// LS Electric XG5000 project: 과년1번패턴
// PLC NewPLC
// module base 0 slot 0: 입출력 모듈:XBC-DR20S (DC 24V 입력 12점, 릴레이 출력 8점)

PROGRAM NewProgram (task: 스캔 프로그램)

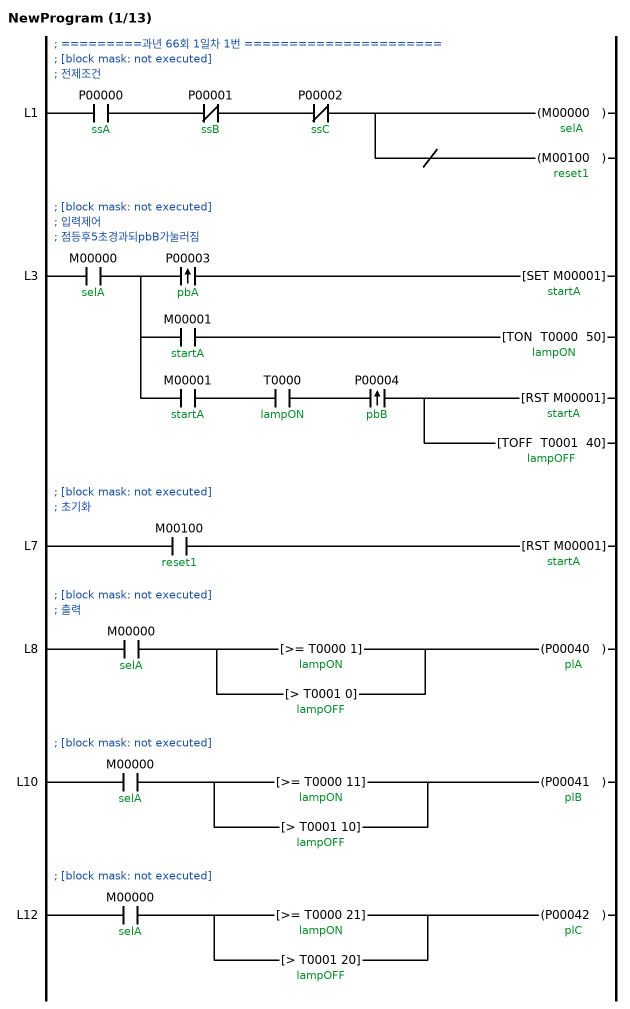
// =========과년 66회 1일차 1번 ======================
; L1 (block mask: not executed)
LOAD      P00000	// ssA
AND NOT   P00001	// ssB
AND NOT   P00002	// ssC
OUT       M00000	// selA
NOT
OUT       M00100	// reset1
// output comment: 전제조건
; L3 (block mask: not executed)
LOAD      M00000	// selA
MPUSH
ANDP      P00003	// pbA
SET       M00001	// startA
MLOAD
AND       M00001	// startA
TON       T0000 50	// lampON
MPOP
AND       M00001	// startA
AND       T0000	// lampON
ANDP      P00004	// pbB
RST       M00001	// startA
TOFF      T0001 40	// lampOFF
// output comment: 입력제어
// output comment: 점등후5초경과되pbB가눌러짐
; L7 (block mask: not executed)
LOAD      M00100	// reset1
RST       M00001	// startA
// output comment: 초기화
; L8 (block mask: not executed)
LOAD      M00000	// selA
LOAD>=    T0000 1	// lampON
OR>       T0001 0	// lampOFF
AND LOAD
OUT       P00040	// plA
// output comment: 출력
; L10 (block mask: not executed)
LOAD      M00000	// selA
LOAD>=    T0000 11	// lampON
OR>       T0001 10	// lampOFF
AND LOAD
OUT       P00041	// plB
; L12 (block mask: not executed)
LOAD      M00000	// selA
LOAD>=    T0000 21	// lampON
OR>       T0001 20	// lampOFF
AND LOAD
OUT       P00042	// plC

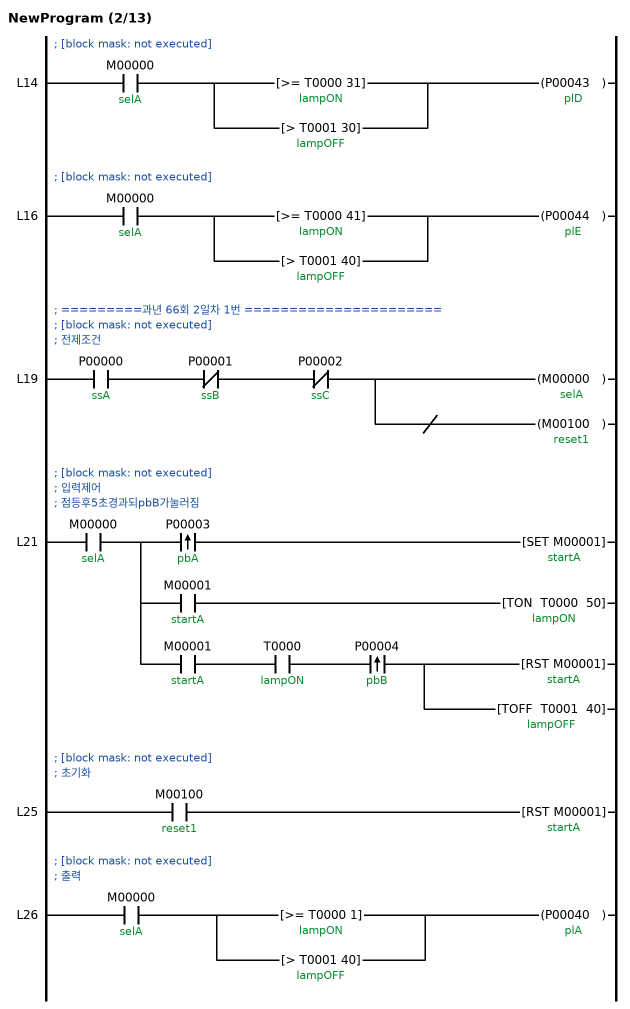
; L14 (block mask: not executed)
LOAD      M00000	// selA
LOAD>=    T0000 31	// lampON
OR>       T0001 30	// lampOFF
AND LOAD
OUT       P00043	// plD
; L16 (block mask: not executed)
LOAD      M00000	// selA
LOAD>=    T0000 41	// lampON
OR>       T0001 40	// lampOFF
AND LOAD
OUT       P00044	// plE
// =========과년 66회 2일차 1번 ======================
; L19 (block mask: not executed)
LOAD      P00000	// ssA
AND NOT   P00001	// ssB
AND NOT   P00002	// ssC
OUT       M00000	// selA
NOT
OUT       M00100	// reset1
// output comment: 전제조건
; L21 (block mask: not executed)
LOAD      M00000	// selA
MPUSH
ANDP      P00003	// pbA
SET       M00001	// startA
MLOAD
AND       M00001	// startA
TON       T0000 50	// lampON
MPOP
AND       M00001	// startA
AND       T0000	// lampON
ANDP      P00004	// pbB
RST       M00001	// startA
TOFF      T0001 40	// lampOFF
// output comment: 입력제어
// output comment: 점등후5초경과되pbB가눌러짐
; L25 (block mask: not executed)
LOAD      M00100	// reset1
RST       M00001	// startA
// output comment: 초기화
; L26 (block mask: not executed)
LOAD      M00000	// selA
LOAD>=    T0000 1	// lampON
OR>       T0001 40	// lampOFF
AND LOAD
OUT       P00040	// plA
// output comment: 출력

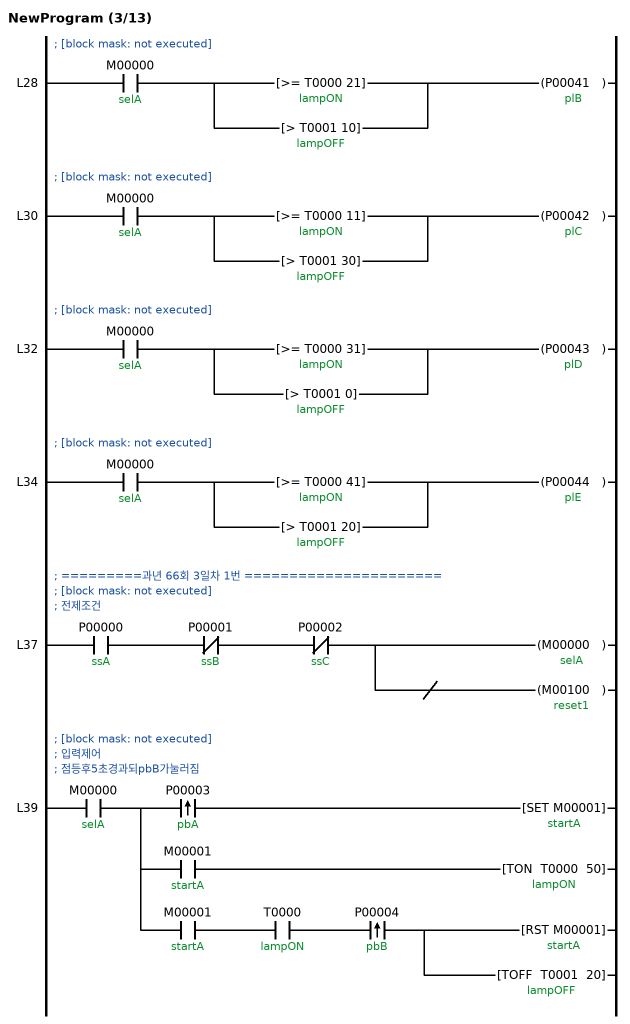
; L28 (block mask: not executed)
LOAD      M00000	// selA
LOAD>=    T0000 21	// lampON
OR>       T0001 10	// lampOFF
AND LOAD
OUT       P00041	// plB
; L30 (block mask: not executed)
LOAD      M00000	// selA
LOAD>=    T0000 11	// lampON
OR>       T0001 30	// lampOFF
AND LOAD
OUT       P00042	// plC
; L32 (block mask: not executed)
LOAD      M00000	// selA
LOAD>=    T0000 31	// lampON
OR>       T0001 0	// lampOFF
AND LOAD
OUT       P00043	// plD
; L34 (block mask: not executed)
LOAD      M00000	// selA
LOAD>=    T0000 41	// lampON
OR>       T0001 20	// lampOFF
AND LOAD
OUT       P00044	// plE
// =========과년 66회 3일차 1번 ======================
; L37 (block mask: not executed)
LOAD      P00000	// ssA
AND NOT   P00001	// ssB
AND NOT   P00002	// ssC
OUT       M00000	// selA
NOT
OUT       M00100	// reset1
// output comment: 전제조건
; L39 (block mask: not executed)
LOAD      M00000	// selA
MPUSH
ANDP      P00003	// pbA
SET       M00001	// startA
MLOAD
AND       M00001	// startA
TON       T0000 50	// lampON
MPOP
AND       M00001	// startA
AND       T0000	// lampON
ANDP      P00004	// pbB
RST       M00001	// startA
TOFF      T0001 20	// lampOFF
// output comment: 입력제어
// output comment: 점등후5초경과되pbB가눌러짐

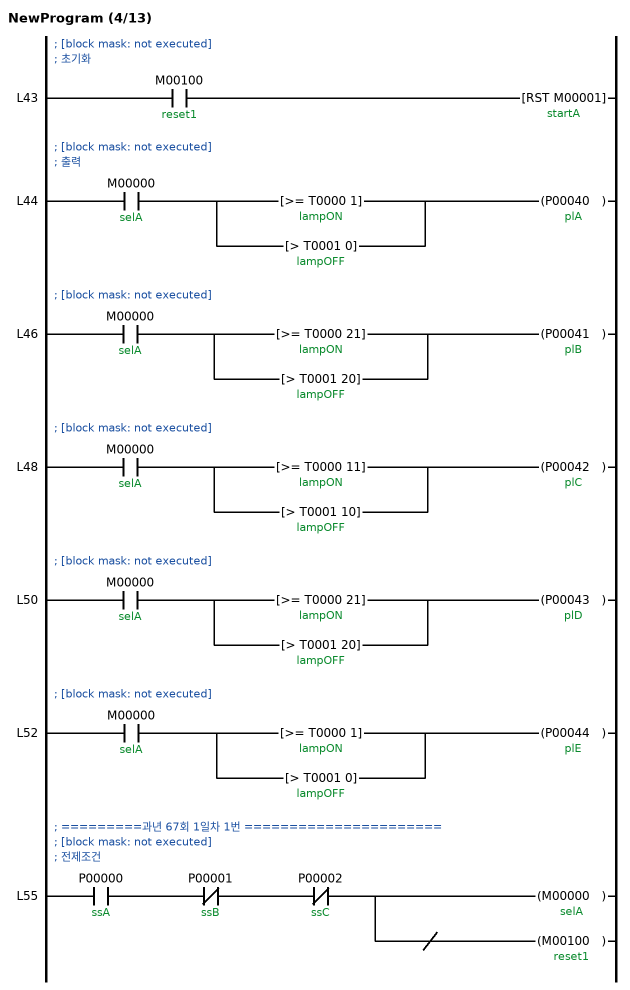
; L43 (block mask: not executed)
LOAD      M00100	// reset1
RST       M00001	// startA
// output comment: 초기화
; L44 (block mask: not executed)
LOAD      M00000	// selA
LOAD>=    T0000 1	// lampON
OR>       T0001 0	// lampOFF
AND LOAD
OUT       P00040	// plA
// output comment: 출력
; L46 (block mask: not executed)
LOAD      M00000	// selA
LOAD>=    T0000 21	// lampON
OR>       T0001 20	// lampOFF
AND LOAD
OUT       P00041	// plB
; L48 (block mask: not executed)
LOAD      M00000	// selA
LOAD>=    T0000 11	// lampON
OR>       T0001 10	// lampOFF
AND LOAD
OUT       P00042	// plC
; L50 (block mask: not executed)
LOAD      M00000	// selA
LOAD>=    T0000 21	// lampON
OR>       T0001 20	// lampOFF
AND LOAD
OUT       P00043	// plD
; L52 (block mask: not executed)
LOAD      M00000	// selA
LOAD>=    T0000 1	// lampON
OR>       T0001 0	// lampOFF
AND LOAD
OUT       P00044	// plE
// =========과년 67회 1일차 1번 ======================
; L55 (block mask: not executed)
LOAD      P00000	// ssA
AND NOT   P00001	// ssB
AND NOT   P00002	// ssC
OUT       M00000	// selA
NOT
OUT       M00100	// reset1
// output comment: 전제조건

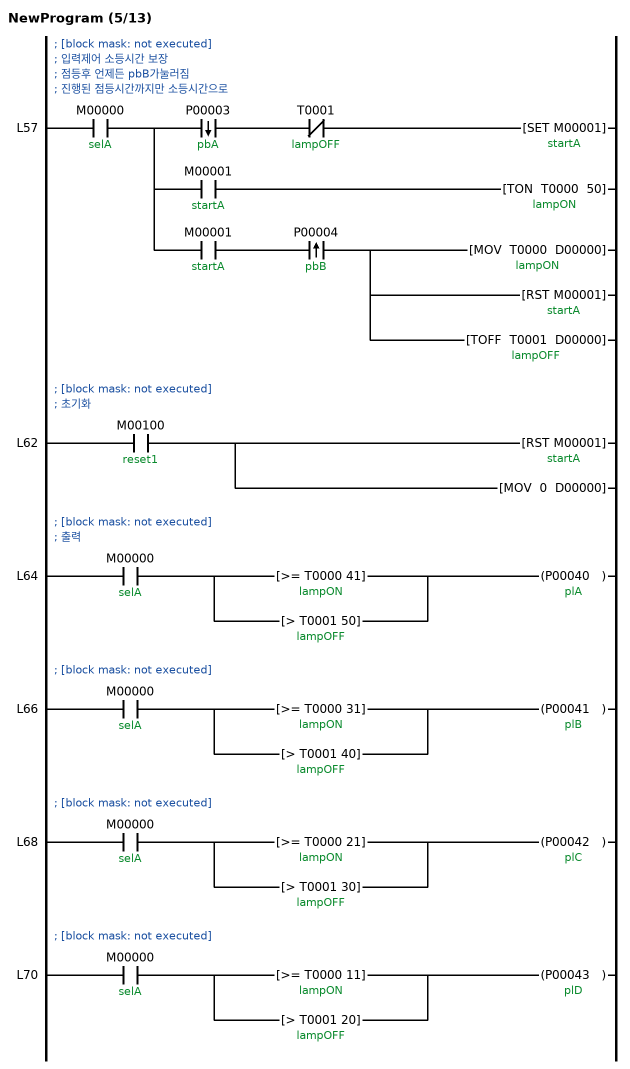
; L57 (block mask: not executed)
LOAD      M00000	// selA
MPUSH
ANDN      P00003	// pbA
AND NOT   T0001	// lampOFF
SET       M00001	// startA
MLOAD
AND       M00001	// startA
TON       T0000 50	// lampON
MPOP
AND       M00001	// startA
ANDP      P00004	// pbB
MOV       T0000 D00000	// lampON
RST       M00001	// startA
TOFF      T0001 D00000	// lampOFF
// output comment: 입력제어 소등시간 보장
// output comment: 점등후 언제든 pbB가눌러짐
// output comment: 
// output comment: 진행된 점등시간까지만 소등시간으로
; L62 (block mask: not executed)
LOAD      M00100	// reset1
RST       M00001	// startA
MOV       0 D00000
// output comment: 초기화
; L64 (block mask: not executed)
LOAD      M00000	// selA
LOAD>=    T0000 41	// lampON
OR>       T0001 50	// lampOFF
AND LOAD
OUT       P00040	// plA
// output comment: 출력
; L66 (block mask: not executed)
LOAD      M00000	// selA
LOAD>=    T0000 31	// lampON
OR>       T0001 40	// lampOFF
AND LOAD
OUT       P00041	// plB
; L68 (block mask: not executed)
LOAD      M00000	// selA
LOAD>=    T0000 21	// lampON
OR>       T0001 30	// lampOFF
AND LOAD
OUT       P00042	// plC
; L70 (block mask: not executed)
LOAD      M00000	// selA
LOAD>=    T0000 11	// lampON
OR>       T0001 20	// lampOFF
AND LOAD
OUT       P00043	// plD

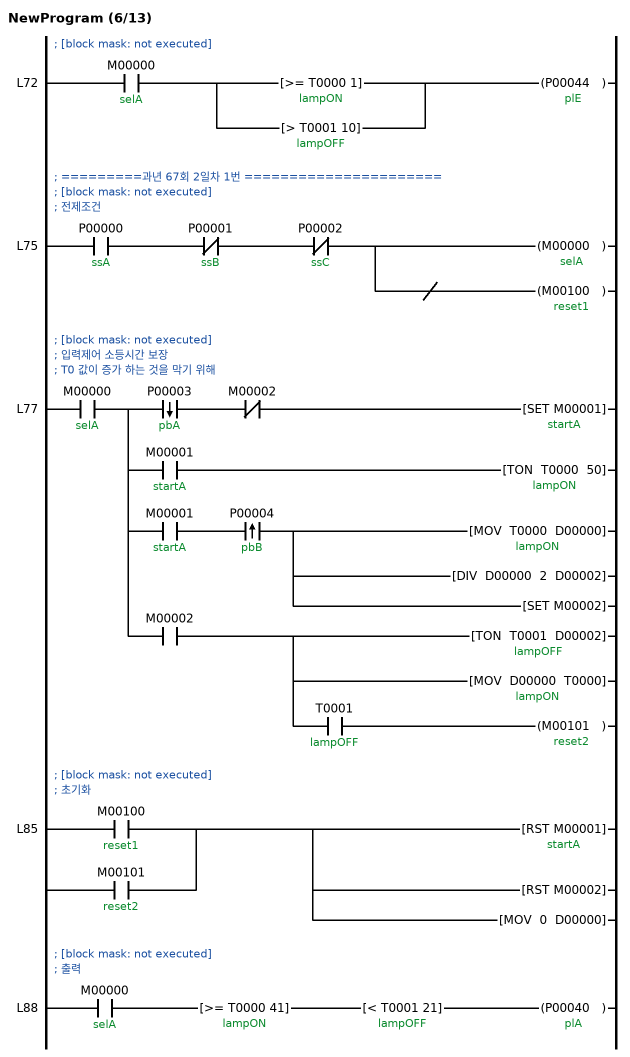
; L72 (block mask: not executed)
LOAD      M00000	// selA
LOAD>=    T0000 1	// lampON
OR>       T0001 10	// lampOFF
AND LOAD
OUT       P00044	// plE
// =========과년 67회 2일차 1번 ======================
; L75 (block mask: not executed)
LOAD      P00000	// ssA
AND NOT   P00001	// ssB
AND NOT   P00002	// ssC
OUT       M00000	// selA
NOT
OUT       M00100	// reset1
// output comment: 전제조건
; L77 (block mask: not executed)
LOAD      M00000	// selA
MPUSH
ANDN      P00003	// pbA
AND NOT   M00002
SET       M00001	// startA
MLOAD
AND       M00001	// startA
TON       T0000 50	// lampON
MLOAD
AND       M00001	// startA
ANDP      P00004	// pbB
MOV       T0000 D00000	// lampON
DIV       D00000 2 D00002
SET       M00002
MPOP
AND       M00002
TON       T0001 D00002	// lampOFF
MOV       D00000 T0000	// lampON
AND       T0001	// lampOFF
OUT       M00101	// reset2
// output comment: 입력제어 소등시간 보장
// output comment: T0 값이 증가 하는 것을 막기 위해
; L85 (block mask: not executed)
LOAD      M00100	// reset1
OR        M00101	// reset2
RST       M00001	// startA
RST       M00002
MOV       0 D00000
// output comment: 초기화
; L88 (block mask: not executed)
LOAD      M00000	// selA
AND>=     T0000 41	// lampON
AND<      T0001 21	// lampOFF
OUT       P00040	// plA
// output comment: 출력

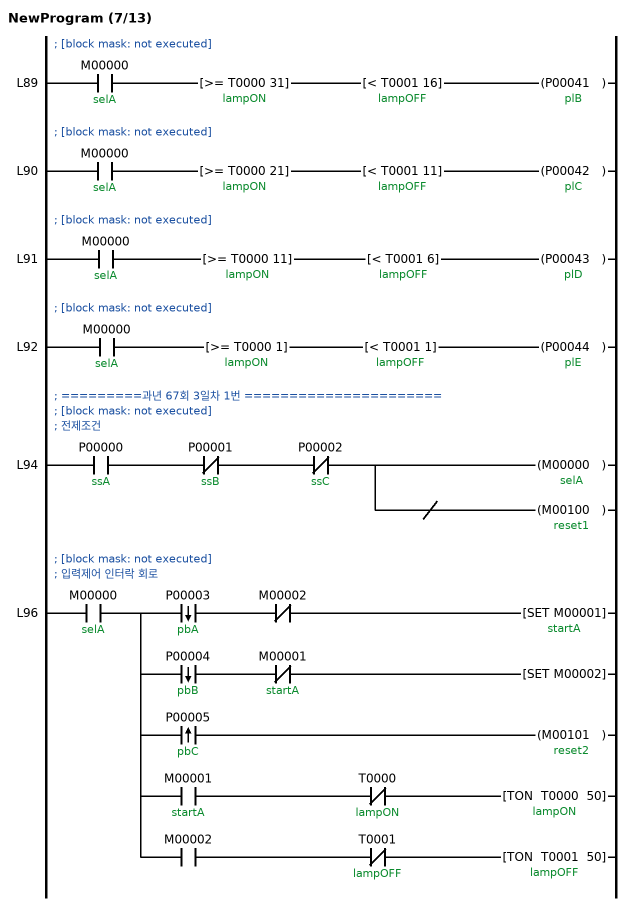
; L89 (block mask: not executed)
LOAD      M00000	// selA
AND>=     T0000 31	// lampON
AND<      T0001 16	// lampOFF
OUT       P00041	// plB
; L90 (block mask: not executed)
LOAD      M00000	// selA
AND>=     T0000 21	// lampON
AND<      T0001 11	// lampOFF
OUT       P00042	// plC
; L91 (block mask: not executed)
LOAD      M00000	// selA
AND>=     T0000 11	// lampON
AND<      T0001 6	// lampOFF
OUT       P00043	// plD
; L92 (block mask: not executed)
LOAD      M00000	// selA
AND>=     T0000 1	// lampON
AND<      T0001 1	// lampOFF
OUT       P00044	// plE
// =========과년 67회 3일차 1번 ======================
; L94 (block mask: not executed)
LOAD      P00000	// ssA
AND NOT   P00001	// ssB
AND NOT   P00002	// ssC
OUT       M00000	// selA
NOT
OUT       M00100	// reset1
// output comment: 전제조건
; L96 (block mask: not executed)
LOAD      M00000	// selA
MPUSH
ANDN      P00003	// pbA
AND NOT   M00002
SET       M00001	// startA
MLOAD
ANDN      P00004	// pbB
AND NOT   M00001	// startA
SET       M00002
MLOAD
ANDP      P00005	// pbC
OUT       M00101	// reset2
MLOAD
AND       M00001	// startA
AND NOT   T0000	// lampON
TON       T0000 50	// lampON
MPOP
AND       M00002
AND NOT   T0001	// lampOFF
TON       T0001 50	// lampOFF
// output comment: 입력제어 인터락 회로

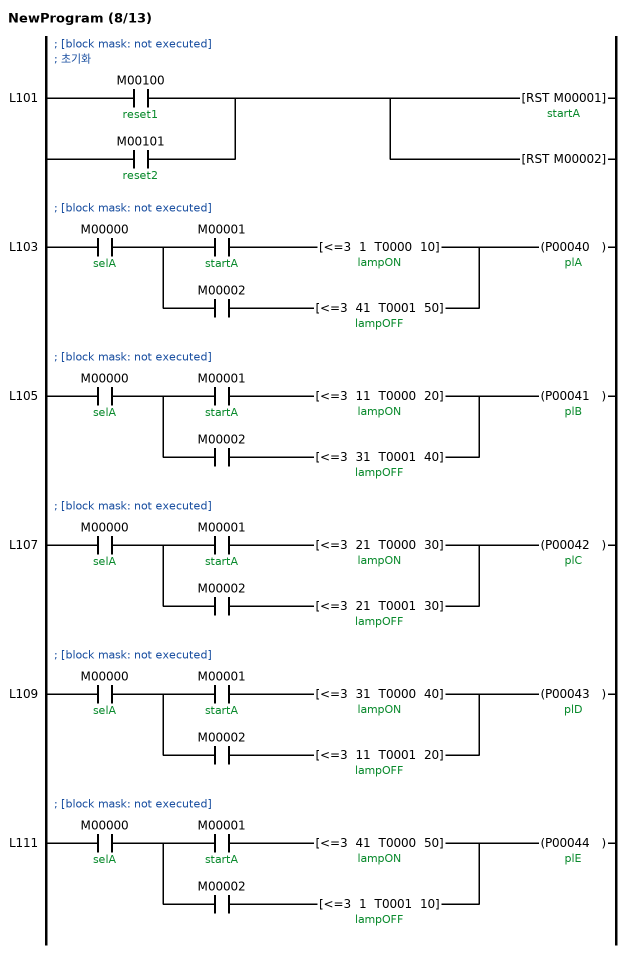
; L101 (block mask: not executed)
LOAD      M00100	// reset1
OR        M00101	// reset2
RST       M00001	// startA
RST       M00002
// output comment: 초기화
; L103 (block mask: not executed)
LOAD      M00000	// selA
LOAD      M00001	// startA
AND<=3    1 T0000 10	// lampON
LOAD      M00002
AND<=3    41 T0001 50	// lampOFF
OR LOAD
AND LOAD
OUT       P00040	// plA
; L105 (block mask: not executed)
LOAD      M00000	// selA
LOAD      M00001	// startA
AND<=3    11 T0000 20	// lampON
LOAD      M00002
AND<=3    31 T0001 40	// lampOFF
OR LOAD
AND LOAD
OUT       P00041	// plB
; L107 (block mask: not executed)
LOAD      M00000	// selA
LOAD      M00001	// startA
AND<=3    21 T0000 30	// lampON
LOAD      M00002
AND<=3    21 T0001 30	// lampOFF
OR LOAD
AND LOAD
OUT       P00042	// plC
; L109 (block mask: not executed)
LOAD      M00000	// selA
LOAD      M00001	// startA
AND<=3    31 T0000 40	// lampON
LOAD      M00002
AND<=3    11 T0001 20	// lampOFF
OR LOAD
AND LOAD
OUT       P00043	// plD
; L111 (block mask: not executed)
LOAD      M00000	// selA
LOAD      M00001	// startA
AND<=3    41 T0000 50	// lampON
LOAD      M00002
AND<=3    1 T0001 10	// lampOFF
OR LOAD
AND LOAD
OUT       P00044	// plE

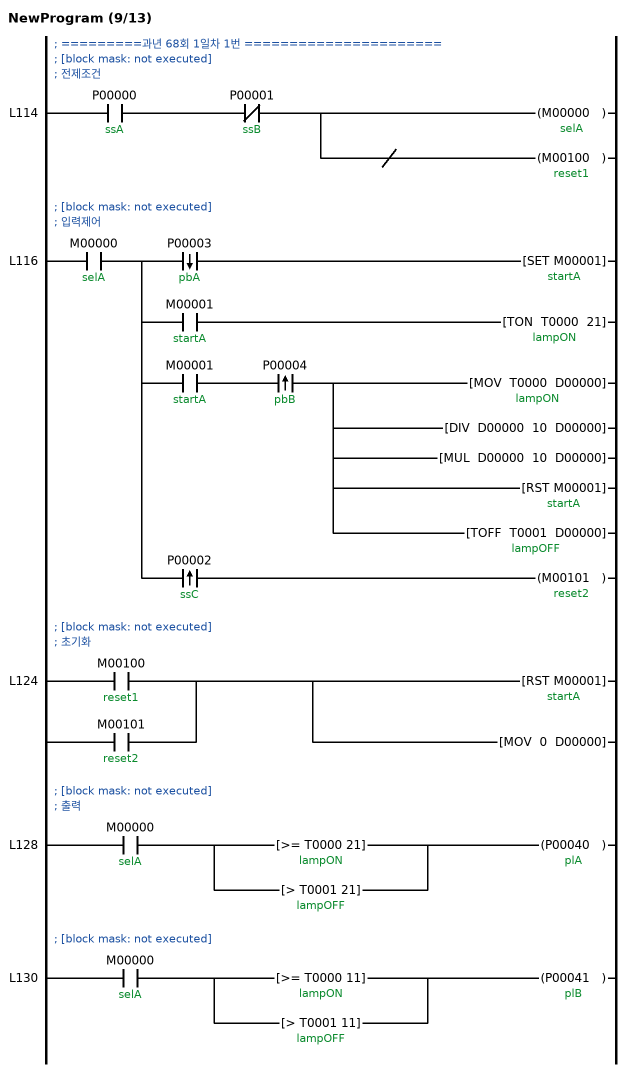
// =========과년 68회 1일차 1번 ======================
; L114 (block mask: not executed)
LOAD      P00000	// ssA
AND NOT   P00001	// ssB
OUT       M00000	// selA
NOT
OUT       M00100	// reset1
// output comment: 전제조건
; L116 (block mask: not executed)
LOAD      M00000	// selA
MPUSH
ANDN      P00003	// pbA
SET       M00001	// startA
MLOAD
AND       M00001	// startA
TON       T0000 21	// lampON
MLOAD
AND       M00001	// startA
ANDP      P00004	// pbB
MOV       T0000 D00000	// lampON
DIV       D00000 10 D00000
MUL       D00000 10 D00000
RST       M00001	// startA
TOFF      T0001 D00000	// lampOFF
MPOP
ANDP      P00002	// ssC
OUT       M00101	// reset2
// output comment: 입력제어
; L124 (block mask: not executed)
LOAD      M00100	// reset1
OR        M00101	// reset2
RST       M00001	// startA
MOV       0 D00000
// output comment: 초기화
; L128 (block mask: not executed)
LOAD      M00000	// selA
LOAD>=    T0000 21	// lampON
OR>       T0001 21	// lampOFF
AND LOAD
OUT       P00040	// plA
// output comment: 출력
; L130 (block mask: not executed)
LOAD      M00000	// selA
LOAD>=    T0000 11	// lampON
OR>       T0001 11	// lampOFF
AND LOAD
OUT       P00041	// plB

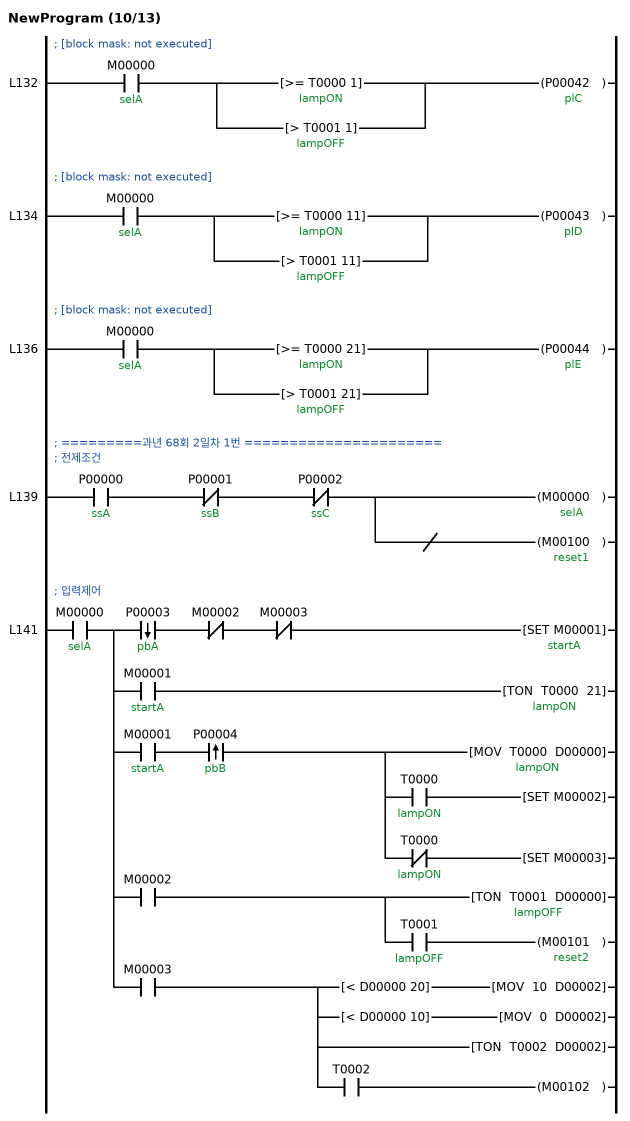
; L132 (block mask: not executed)
LOAD      M00000	// selA
LOAD>=    T0000 1	// lampON
OR>       T0001 1	// lampOFF
AND LOAD
OUT       P00042	// plC
; L134 (block mask: not executed)
LOAD      M00000	// selA
LOAD>=    T0000 11	// lampON
OR>       T0001 11	// lampOFF
AND LOAD
OUT       P00043	// plD
; L136 (block mask: not executed)
LOAD      M00000	// selA
LOAD>=    T0000 21	// lampON
OR>       T0001 21	// lampOFF
AND LOAD
OUT       P00044	// plE
// =========과년 68회 2일차 1번 ======================
; L139
LOAD      P00000	// ssA
AND NOT   P00001	// ssB
AND NOT   P00002	// ssC
OUT       M00000	// selA
NOT
OUT       M00100	// reset1
// output comment: 전제조건
; L141
LOAD      M00000	// selA
MPUSH
ANDN      P00003	// pbA
AND NOT   M00002
AND NOT   M00003
SET       M00001	// startA
MLOAD
AND       M00001	// startA
TON       T0000 21	// lampON
MLOAD
AND       M00001	// startA
ANDP      P00004	// pbB
MOV       T0000 D00000	// lampON
MPUSH
AND       T0000	// lampON
SET       M00002
MPOP
AND NOT   T0000	// lampON
SET       M00003
MLOAD
AND       M00002
TON       T0001 D00000	// lampOFF
AND       T0001	// lampOFF
OUT       M00101	// reset2
MPOP
AND       M00003
MPUSH
AND<      D00000 20
MOV       10 D00002
MLOAD
AND<      D00000 10
MOV       0 D00002
MPOP
TON       T0002 D00002
AND       T0002
OUT       M00102
// output comment: 입력제어

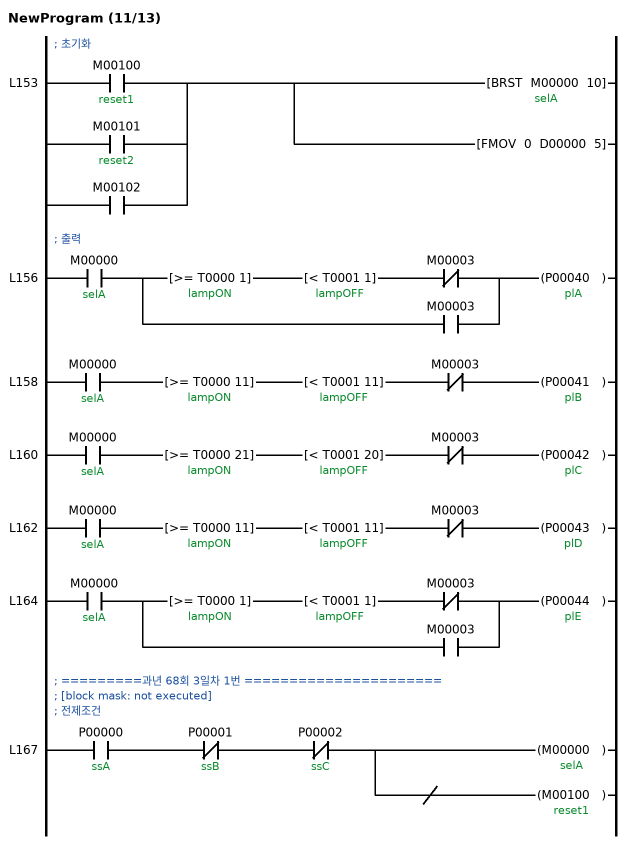
; L153
LOAD      M00100	// reset1
OR        M00101	// reset2
OR        M00102
BRST      M00000 10	// selA
FMOV      0 D00000 5
// output comment: 초기화
; L156
LOAD      M00000	// selA
LOAD>=    T0000 1	// lampON
AND<      T0001 1	// lampOFF
AND NOT   M00003
OR        M00003
AND LOAD
OUT       P00040	// plA
// output comment: 출력
; L158
LOAD      M00000	// selA
AND>=     T0000 11	// lampON
AND<      T0001 11	// lampOFF
AND NOT   M00003
OUT       P00041	// plB
; L160
LOAD      M00000	// selA
AND>=     T0000 21	// lampON
AND<      T0001 20	// lampOFF
AND NOT   M00003
OUT       P00042	// plC
; L162
LOAD      M00000	// selA
AND>=     T0000 11	// lampON
AND<      T0001 11	// lampOFF
AND NOT   M00003
OUT       P00043	// plD
; L164
LOAD      M00000	// selA
LOAD>=    T0000 1	// lampON
AND<      T0001 1	// lampOFF
AND NOT   M00003
OR        M00003
AND LOAD
OUT       P00044	// plE
// =========과년 68회 3일차 1번 ======================
; L167 (block mask: not executed)
LOAD      P00000	// ssA
AND NOT   P00001	// ssB
AND NOT   P00002	// ssC
OUT       M00000	// selA
NOT
OUT       M00100	// reset1
// output comment: 전제조건

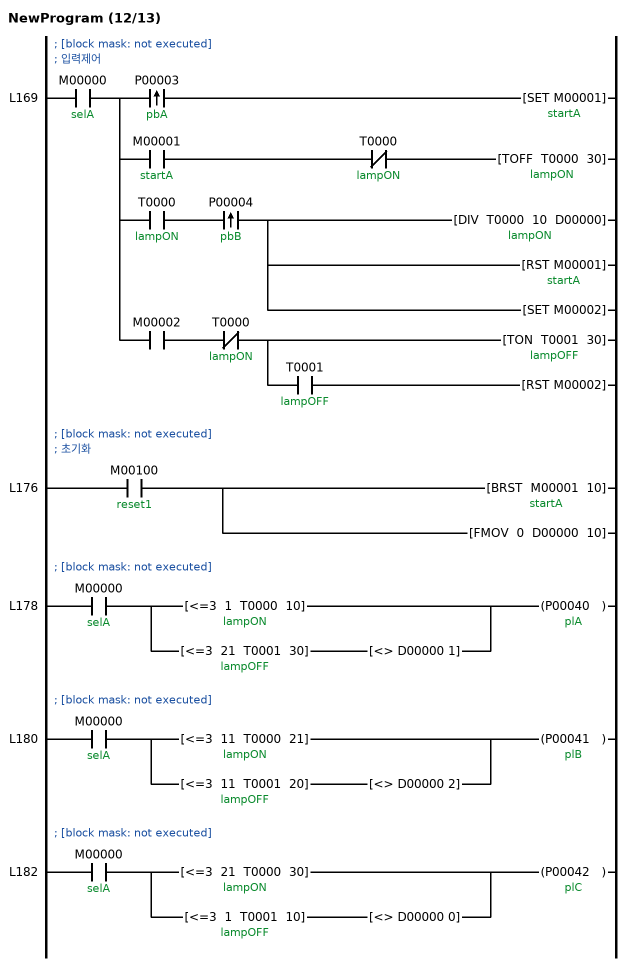
; L169 (block mask: not executed)
LOAD      M00000	// selA
MPUSH
ANDP      P00003	// pbA
SET       M00001	// startA
MLOAD
AND       M00001	// startA
AND NOT   T0000	// lampON
TOFF      T0000 30	// lampON
MLOAD
AND       T0000	// lampON
ANDP      P00004	// pbB
DIV       T0000 10 D00000	// lampON
RST       M00001	// startA
SET       M00002
MPOP
AND       M00002
AND NOT   T0000	// lampON
TON       T0001 30	// lampOFF
AND       T0001	// lampOFF
RST       M00002
// output comment: 입력제어
; L176 (block mask: not executed)
LOAD      M00100	// reset1
BRST      M00001 10	// startA
FMOV      0 D00000 10
// output comment: 초기화
; L178 (block mask: not executed)
LOAD      M00000	// selA
LOAD<=3   1 T0000 10	// lampON
LOAD<=3   21 T0001 30	// lampOFF
AND<>     D00000 1
OR LOAD
AND LOAD
OUT       P00040	// plA
; L180 (block mask: not executed)
LOAD      M00000	// selA
LOAD<=3   11 T0000 21	// lampON
LOAD<=3   11 T0001 20	// lampOFF
AND<>     D00000 2
OR LOAD
AND LOAD
OUT       P00041	// plB
; L182 (block mask: not executed)
LOAD      M00000	// selA
LOAD<=3   21 T0000 30	// lampON
LOAD<=3   1 T0001 10	// lampOFF
AND<>     D00000 0
OR LOAD
AND LOAD
OUT       P00042	// plC

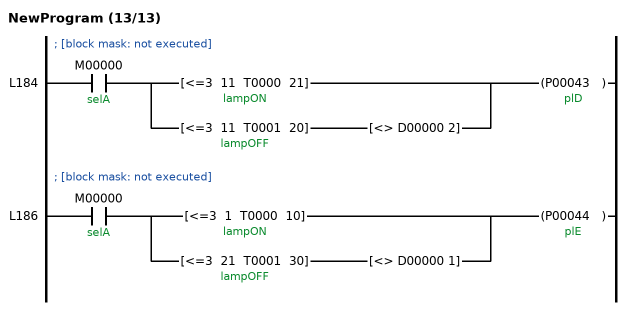
; L184 (block mask: not executed)
LOAD      M00000	// selA
LOAD<=3   11 T0000 21	// lampON
LOAD<=3   11 T0001 20	// lampOFF
AND<>     D00000 2
OR LOAD
AND LOAD
OUT       P00043	// plD
; L186 (block mask: not executed)
LOAD      M00000	// selA
LOAD<=3   1 T0000 10	// lampON
LOAD<=3   21 T0001 30	// lampOFF
AND<>     D00000 1
OR LOAD
AND LOAD
OUT       P00044	// plE